// TIA Portal V20 export
TYPE "typeCmControlNodeCommand"
// stored: Namespace Unit1.Em2
   STRUCT
      jrOutPnPLeftAxisX : "LER_typeAxisCommand";
      jrOutPnPLeftAxisZ : "LER_typeAxisCommand";
      jrOutPnPRightAxisX : "LER_typeAxisCommand";
      jrOutPnPRightAxisZ : "LER_typeAxisCommand";
      jrOutPnPLeftClamp : "LER_typeTwoWayActCommand";
      jrOutPnPRightClamp : "LER_typeTwoWayActCommand";
   END_STRUCT;
END_TYPE
